(* IEC 61131-3 sources: blark/blark/tests/source, 15 files *)

(* ---- commas_in_case.st ---- *)
(*<textarea rows="15" cols="81">
********************************************************************************
* Comments
********************************************************************************
</textarea>*)
FUNCTION fun_CommainCase : BOOL
VAR_INPUT
    (* Byte to be evaluated as a printable character. *)
    character : BYTE;
END_VAR

CASE character OF
    (*
    Any character that falls in the ascii range (in base-10)
    0-8, 11, 12, 14-27 or >=127 is an invalid character.
    *)
    BYTE#9..BYTE#10, BYTE#13, BYTE#28..BYTE#126:
        fun_CommainCase := TRUE;
ELSE
    fun_CommainCase := FALSE;
END_CASE
END_FUNCTION

(* ---- pointer_fb_initialized.st ---- *)
FUNCTION dummyFunction : BOOL
VAR_INPUT
     pt_SomethingNeat : POINTER TO struct_SomethingNeat;
     pt_CrossTaskWriter : POINTER TO fb_crossTaskWrite(ID := gvl_mutexId.MUTEX_ONE, sizeOfStruct := SIZEOF(DINT));
     pt_CrossTaskWriter : POINTER TO fb_crossTaskWrite(ID := gvl_mutexId.MUTEX_TWO, sizeOfStruct := SIZEOF(quality_t));
END_VAR
END_FUNCTION

(* ---- array_of_addresses.st ---- *)
FUNCTION_BLOCK class_SomethingCool
VAR
        currentChannel : ARRAY[1..g_c_someConstant] OF POINTER TO struct_groupData :=
                [       ADR(_object[1].someValue),
                        ADR(_object[2].someValue),
                        ADR(_object[3].someValue),
                        ADR(_object[4].someValue),
                        ADR(_object[5].someValue),
                        ADR(_object[6].someValue),
                        ADR(_object[7].someValue),
                        ADR(_object[8].someValue),
                        ADR(_object[9].someValue),
                        ADR(_object[10].someValue)
                ];
END_VAR
END_FUNCTION_BLOCK

(* ---- fb_w_public_access.st ---- *)
FUNCTION_BLOCK PUBLIC class_PublicFB
    VAR_OUTPUT
        (*Some comment.*)
        Error     : BOOL;
    END_VAR
END_FUNCTION_BLOCK

(* ---- pointer_to_pointer_to.st ---- *)
FUNCTION_BLOCK fb_test
    VAR
        _pt_Strings : POINTER TO POINTER TO someObject;
        _pt_Current : POINTER TO POINTER TO someObject;
    END_VAR
END_FUNCTION_BLOCK

(* ---- type_and_fb.st ---- *)
TYPE
    color: (red, green, blue);
END_TYPE

FUNCTION_BLOCK Testblock
    VAR_INPUT
        number_of_boxes: INT;
    END_VAR
    VAR
        cabinet: color;
    END_VAR

    IF number_of_boxes > 1 THEN
        cabinet := green;
    END_IF
END_FUNCTION_BLOCK

(* ---- and_then_or_else.st ---- *)
(*<textarea rows="15" cols="81">
********************************************************************************
**** a great, big, long multiline comment
********************************************************************************
</textarea>*)
METHOD Split : POINTER TO STRING (*Returns a pointer to an error string.
Returns zero on success.*)
VAR_IN_OUT
    (* The class_SELString containing the combination of characters to denote
the locations where the split shall occur.*)
    sep    : class_Object;
END_VAR

IF TestOne AND_THEN TestTwo THEN
    DoSomething();
ELSIF TestThree OR_ELSE TestFour THEN
    DoSomethingElse();
END_IF

END_METHOD

(* ---- array_initializer.st ---- *)
(* This program creates an array of objects using array initialization. *)
PROGRAM oop_test
VAR
    runners : ARRAY[RunnerTasks.RUNNER_START+1..RunnerTasks.RUNNER_END-1] OF FB_Runner[
        (instanceName := 'one'),
        (instanceName := 'two'),
        (instanceName := 'three'),
        (instanceName := 'four'),
        (instanceName := 'five'),
        (instanceName := 'six'),
        (instanceName := 'seven'),
        (instanceName := 'eight'),
        (instanceName := 'nine'),
        (instanceName := 'ten'),
        (instanceName := 'elevin'),
        (instanceName := 'thirteen'),
        (instanceName := 'fourteen'),
        (instanceName := 'fifteen'),
        (instanceName := 'sixteen'),
        (instanceName := 'seventeen'),
        (instanceName := 'eighteen')
    ];
    aSample   : ARRAY[1..2] OF FB_Sample[(nInitParam := 4), (nInitParam := 7)]
                            := [(nInput := 5, nMyProperty := 6), (nInput := 8, nMyProperty := 9)];
END_VAR

END_PROGRAM

(* ---- array_of_arrays.st ---- *)
{attribute 'hide'}
METHOD prv_Detection : BOOL
VAR_IN_OUT
        currentChannel : ARRAY[APhase..CPhase] OF ARRAY [1..5] OF INT := [
                [1, 2, 3, 4, 5],
                [1, 2, 3, 4, 5],
                [1, 2, 3, 4, 5]
        ];
END_VAR

// do some stuff
END_METHOD

(* ---- array_of_objects.st ---- *)
{attribute 'hide'}
METHOD prv_Detection : BOOL
VAR_IN_OUT
        currentChannel : ARRAY[APhase..CPhase] OF class_baseVector(SIZEOF(vector_t),0);
END_VAR

// do some stuff
END_METHOD

(* ---- array_with_integer_initializer.st ---- *)
{attribute 'hide'}
METHOD prv_Detection : BOOL
VAR_IN_OUT
        currentChannel : ARRAY[*] OF someStruct := 0;
END_VAR

// do some stuff
END_METHOD

(* ---- dereference_method.st ---- *)
METHOD DoSomething
VAR
    Something : BOOL;
END_VAR

Something := anObject.WriteLine(THIS^.something.t, THIS^.GetTagName()^, INT_TO_STRING(BOOL_TO_INT(THIS^.someAttribute)));

END_METHOD

(* ---- fb_initializer.st ---- *)
(* This program creates a function block instance with initialization. *)
PROGRAM oop_test
VAR
    fbSample  : FB_Sample(nInitParam := 1) := (nInput := 2, nMyProperty := 3);
END_VAR

END_PROGRAM

(* ---- object_oriented_dotaccess.st ---- *)
(* This program uses some object-oriented function-block with multiline access. *)
PROGRAM oop_test
VAR
        uut : SomeFunctionBlock;
END_VAR

// Use an object that has a different method called on each line
uut.DoSomething(input_1:='foo', input_2:='bar')
   .DoSomethingElse(input_1:=5)
   .Finish();

// Or perhaps something that's a little more tame
uut.DoSomething(input_1:='foo', input_2:='bar')
   .DoSomethingElse(input_1:=5).Finish();

// Or something tamer, still
uut.DoSomething(input_1:='foo', input_2:='bar').DoSomethingElse(input_1:=5).Finish();

END_PROGRAM

(* ---- stray_comment.st ---- *)
(* Call this method to truncate an LREAL value *);
{attribute 'hide'}
METHOD prv_Floor : LREAL
VAR_INPUT
        Input : LREAL;
END_VAR
VAR
        Round : LINT;
END_VAR
Round := LREAL_TO_LINT(Input);
IF LINT_TO_LREAL(Round) <= Input THEN
        prv_Floor := LINT_TO_LREAL(Round);
ELSE
        prv_Floor := LINT_TO_LREAL(Round - 1);
END_IF
END_METHOD
